(* IEC 61131-3 sources: 89152_FlorisHendrix_AfstudeerProject/89152_FlorisHendrix_ExamenProject/Stations/MachineControl/MachineControl/Class/StringRAM, 1 file *)

(* ---- StringRAM.st ---- *)
(*!
<Class
	Name               = "StringRAM"
	Revision           = "1.10"
	RealtimeTask       = "false"
	CyclicTask         = "false"
	BackgroundTask     = "false"
	Sigmatek           = "true"
	OSInterface        = "false"
	HighPriority       = "false"
	Automatic          = "false"
	UpdateMode         = "Prescan"
	SharedCommandTable = "true"
	Objectsize         = "(420,120)"
	Comment            = "handles character strings, stores data retentive">
	<Channels>
		<Server
			Name           = "Data"
			Initialize     = "true"
			Visualized     = "true"
			WriteProtected = "false">
		</Server>
		<Client Name="DataBuffer" Required="false" Internal="true"/>
		<Client Name="UseFile" Required="false" Internal="false" Comment="init value&#13;&#10;1..RamData is written to file"/>
	</Channels>
	<RevDoku>
		<Owner Company="Sigmatek GmbH"/>
		<Dokumentation Revision="1.10" Date="2012-11-05" Author="spimar" Company="Sigmatek GmbH" Description="New client (SingleRealloc) which is used for an optimized memory handling!"/>
		<Dokumentation Revision="1.2" Date="2012-06-15" Author="feshar" Company="Sigmatek GmbH" Description="Class can use file storage now. (Set The client UseFile to &apos;1&apos;)&#13;&#10;!! If the class is using file storage please note the method UpdateToFile !!"/>
		<Dokumentation Revision="1.1" Date="2011-12-20" Author="spimar" Company="Sigmatek GmbH" Description="Embedded RAMex object is not longer visualized;"/>
	</RevDoku>
	<Network Name="StringRAM">
		<!-- List of Components in this network -->
		<Components>
			<Object
				Name       = "_base"
				Class      = "StringInternal"
				Position   = "(660,240)"
				Visualized = "true">
				<Channels>
					<Server Name="Data"/>
					<Client Name="DataBuffer"/>
					<Client Name="SingleRealloc" Value="1"/>
				</Channels>
			</Object>
			<Object
				Name       = "DataBuffer"
				Class      = "RAMex"
				Position   = "(240,240)"
				Visualized = "false">
				<Channels>
					<Server Name="m_udLength"/>
					<Client Name="MultiTask"/>
					<Client Name="ThreadSafe" Value="0"/>
					<Client Name="UseFile"/>
				</Channels>
			</Object>
		</Components>
		<Comments>
		</Comments>
		<!-- List of Connections in this network -->
		<Connections>
			<Connection Source="_base.DataBuffer" Destination="DataBuffer.m_udLength" Vertices="(660,330),(540,330),"/>
			<Connection Source="this.Data" Destination="_base.Data" Vertices="(1132,210),(960,330),"/>
			<Connection Source="DataBuffer.UseFile" Destination="this.UseFile" Vertices="(240,390),(38,270),"/>
			<Connection Source="_base.SingleRealloc" Destination="this.SingleRealloc" Vertices="(660,390),(600,390),(600,360),(630,300),(600,300),(600,210),(38,210),"/>
		</Connections>
		<!-- Headerfiles -->
		<Options>
		</Options>
	</Network>
</Class>
*)
#pragma using StringInternal

StringRAM : CLASS
: StringInternal
  //Servers:
  //Clients:
	virtual DataBuffer 	: CltChCmd_RAMex;
	UseFile 	: CltCh_DINT;
  //Variables:
  //Functions:
  //Tables:
	FUNCTION @STD
		VAR_OUTPUT
			ret_code	: CONFSTATES;
		END_VAR;
	FUNCTION GLOBAL TAB @CT_;
END_CLASS;

#pragma using RAMex
